TYPE ST_CYLINDER_TagID :
STRUCT
	sDeviceTagID			: STRING(10);
	sRetractTagID			: STRING(10);
	sExtendTagID			: STRING(10);

END_STRUCT
END_TYPE

(* stored: Version 1.1.0.1, ProductVersion 3.1.4024.15
   DUT ST_CYLINDER_TagID: Id {f578e442-587f-4a61-b08d-84f823fb53fa} *)
